(* IEC 61131-3 sources: dynamics/src/TimeProviders, 3 files *)

(* ---- IElapsedSecondsProvider.st ---- *)
NAMESPACE Simatic.Ax.Dynamics
    /// `GetElapsedSeconds` and `Start`
    INTERFACE IElapsedSecondsProvider

        /// Get elapsed time since last call of `Start`
        METHOD GetElapsedSeconds : LREAL END_METHOD

        /// Start time measurement
        METHOD Start END_METHOD

    END_INTERFACE
END_NAMESPACE

(* ---- ConstantTimeProvider.st ---- *)
NAMESPACE Simatic.Ax.Dynamics
    /// Constantly returns `seconds` whenever `GetElapsedSeconds` is called
    CLASS ConstantTimeProvider IMPLEMENTS IElapsedSecondsProvider

        VAR PUBLIC
            /// This value is retured by `GetElapsedSeconds`
            seconds : LREAL;
        END_VAR

        METHOD PUBLIC GetElapsedSeconds : LREAL
            GetElapsedSeconds := seconds;
        END_METHOD

        METHOD PUBLIC Start
            ; // Nothing happens -- that's why it's called constant
        END_METHOD

END_CLASS
END_NAMESPACE

(* ---- MeasuredTimeProvider.st ---- *)
USING Siemens.Simatic.S71500.Clocks;
NAMESPACE Simatic.Ax.Dynamics
    /// Uses a `Siemens.Simatic.S71500.Clocks.RuntimeMeasurement`
    CLASS MeasuredTimeProvider IMPLEMENTS IElapsedSecondsProvider

        VAR PRIVATE
            _measurement : RuntimeMeasurement;
        END_VAR

        METHOD PUBLIC GetElapsedSeconds : LREAL
            GetElapsedSeconds := _measurement.GetElapsedSeconds();
        END_METHOD

        METHOD PUBLIC Start
            _measurement.Start();
        END_METHOD

    END_CLASS
END_NAMESPACE
